# EPICS substitutions: NucInstDigApp/Db/NucInstDigTrace.substitutions
global { "P=\$(P)", "Q=\$(Q)" }

file "NucInstDigTrace.template" {
    pattern { N }
    { "1" }
    { "2" }
    { "3" }
    { "4" }
}
